(* CODESYS project XLH_base_START_01_00.project
   Description: Receives some incoming messages and echoes them with CAN-ID +1
   Title: CAN Bus API Example
   Version: 1.0.0.0
   Company: 3S - Smart Software Solutions GmbH
   Author: 3S - Smart Software Solutions GmbH

Project tree, tasks and I/O mapping:
  XLH_base : CODESYS Control for Raspberry Pi SL, CODESYS, order no. 2302000009, version 4.12.0.0
    application app
      libraries: Standard, 3.5.18.0 (System); Memory, * (3S - Smart Software Solutions GmbH); Util, 3.5.19.0 (System); VisuDialogs, * (System); CAA Tick Extern, 3.5.17.0 (CAA Technical Workgroup); SysTime, 3.5.17.0 (System); CmpIecTask, * (System); xemax Bibliothek, 0.10 (xemax ag)
      task MAIN_TASK (cyclic, interval 20 ms, priority 0) calls MAIN, io
      task VISU_TASK (cyclic, interval 100 ms, priority 31) calls VisuElems.Visu_Prg
      program io [ST]
      visualisation VISU
      program MAIN [ST]
    SoftMotion General Axis Pool
    GPIOs_A_B : GPIOs B+/Pi2, CODESYS, version 4.12.0.0
        input  app.io.bSw1 : BOOL  // digital inputs (GPIO0..GPIO31).Bit4
        input  app.io.bSw2 : BOOL  // digital inputs (GPIO0..GPIO31).Bit5
        input  app.io.bSw3 : BOOL  // digital inputs (GPIO0..GPIO31).Bit6
        input  app.io.bSw4 : BOOL  // digital inputs (GPIO0..GPIO31).Bit12
        input  app.io.bSw5 : BOOL  // digital inputs (GPIO0..GPIO31).Bit13
        input  app.io.bSw6 : BOOL  // digital inputs (GPIO0..GPIO31).Bit16
        input  app.io.bSw7 : BOOL  // digital inputs (GPIO0..GPIO31).Bit17
        input  app.io.bSw8 : BOOL  // digital inputs (GPIO0..GPIO31).Bit19
        output app.io.bLed1 : BOOL  // digital outputs (GPIO0..GPIO31).Bit20
        output app.io.bLed2 : BOOL  // digital outputs (GPIO0..GPIO31).Bit21
        output app.io.bLed3 : BOOL  // digital outputs (GPIO0..GPIO31).Bit22
        output app.io.bLed4 : BOOL  // digital outputs (GPIO0..GPIO31).Bit23
        output app.io.bLed5 : BOOL  // digital outputs (GPIO0..GPIO31).Bit24
        output app.io.bLed6 : BOOL  // digital outputs (GPIO0..GPIO31).Bit26
        output app.io.bLed7 : BOOL  // digital outputs (GPIO0..GPIO31).Bit27
        unmapped channels: digital inputs (GPIO0..GPIO31), digital outputs (GPIO0..GPIO31)
    Onewire
    Camera device
      <Leer>
    SPI
    I²C
    Ethernet : Ethernet, CODESYS, version 4.2.0.0
        settings: IPAddress = [127,0,0,1]; SubnetMask = [255,0,0,0]; GatewayAddress = [0,0,0,0]; NetworkInterfaceName = 'lo'; NetworkInterfaceName = "lo"; SaveCommunicationSettings = FALSE
      ModbusTCP_Slave_OLED_Port_503 : ModbusTCP Slave Device, CODESYS, version 4.3.0.0
          settings: Port = 503
          output app.io.oled.awToOled : ARRAY[0..32] OF WORD  // Ausgänge
          unmapped channels: Eingänge
  libraries: VisuSymbols, 4.5.0.0 (System); DepictorBase, 1.0.5.0 (3S - Smart Software Solutions GmbH)
  text list GlobalTextList
*)

// XLH_base/app/MAIN
PROGRAM MAIN
VAR
	vVersionPlc: VERSION;
	sVersionPlc: STRING(255);
	vVersionLib: VERSION;
	sVersionLib: STRING(255);
END_VAR

// Version Bibliothex xemax
vVersionPlc.uiMajor := 1;
vVersionPlc.uiMinor := 0;
sVersionPlc := CONCAT(TO_STRING(TO_UINT(vVersionPlc.uiMajor)), CONCAT('.', (TO_STRING(TO_UINT(vVersionPlc.uiMinor)))));
vVersionLib := xemax.GetLibVersion();
sVersionLib := CONCAT(TO_STRING(TO_UINT(vVersionLib.uiMajor)), CONCAT('.', (TO_STRING(TO_UINT(vVersionLib.uiMinor)))));

(*
==================================================================================================
Login Codesys in die XLH - SPS 
user: pi
pw: pi
==================================================================================================
Webvisualisierung
http://ip:8080/webvisu.htm
- bei einer Verbindung via USB: http://192.168.31.31:8080/webvisu.htm
- bei einer Verbindung via USB-RJ45-Adapter: http://192.168.1.31:8080/webvisu.htm
==================================================================================================
OPC-UA
anonymous (ohne Benutzer und Passwort)
opc.tcp://192.168.31.31:4840
==================================================================================================
RGB-Matrix
im aktuellen BETA-Status kann die Matrix via REST-API angesteurt werden
https://de.wikipedia.org/wiki/Representational_State_Transfer
http://192.168.1.31:8077/rgb/0/1/0

Weiter geplant ist eine Umsetzung zur Ansteuerung der RGB Matrix als IoT Device via MQTT
 
Die Integration in Codesys ist noch ausstehend 
==================================================================================================
Login XLH - Linuxumgebung via Putty
user: pi
pw: pi
==================================================================================================
Konfiguration WiFi 
sudo nano /etc/wpa_supplicant/wpa_supplicant.conf

network={
        ssid="abc"
        psk="def"
        key_mgmt=WPA-PSK
}
==================================================================================================
statische IP USB-Ethernet-Erweiterung: 
sudo nano /etc/dhcpcd.conf
# profile static_eth0
...
==================================================================================================
*)

END_PROGRAM

// XLH_base/app/io
PROGRAM io
VAR_INPUT			
	bLed1: BOOL;
	bLed2: BOOL;
	bLed3: BOOL;
	bLed4: BOOL;
	bLed5: BOOL;
	bLed6: BOOL;
	bLed7: BOOL;	
	oled: OLED;
END_VAR
VAR_OUTPUT
	bSw1: BOOL;
	bSw2: BOOL;
	bSw3: BOOL;
	bSw4: BOOL;
	bSw5: BOOL;
	bSw6: BOOL;
	bSw7: BOOL;
	bSw8: BOOL;
END_VAR
VAR
END_VAR

xemax.LOCAL_TIME_AND_TIME_ZONE();
xemax.TASK_INFO();
oled();

END_PROGRAM

// XLH_base/app/VISU
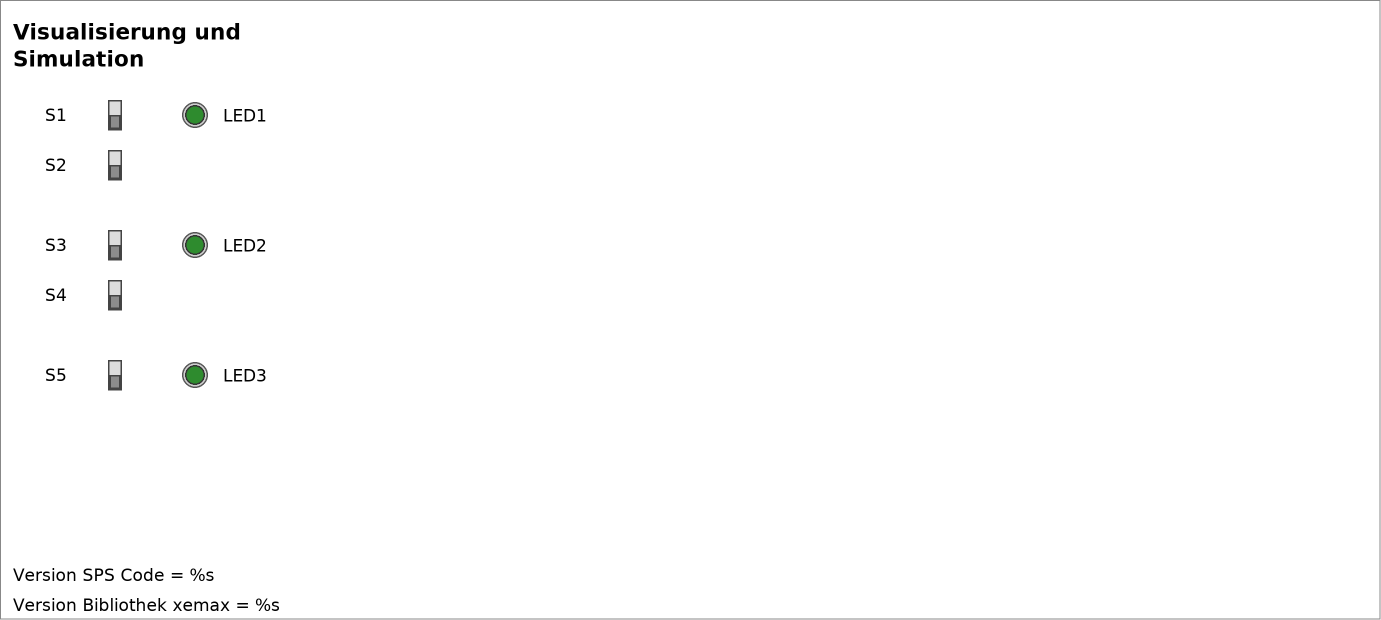
VISUALIZATION VISU  // 1381x620
    Rectangle (220,90 81x51), "LED1"
    Rectangle (10,10 461x71), "Visualisierung und Simulation"
    Line (1380,270)
    DipSwitch (80,100 70x30), variable: io.bSw1, behaviour: TOGGLE, style: Switch-DipSwitch-Gray
    Rectangle (20,90 50x50), "S1"
    Lamp1 (180,100 30x30), variable: io.bLed1, style: Lamp-Lamp1-Green
    Rectangle (10,560 291x30), "Version SPS Code = %s", text variable: MAIN.sVersionPlc
    Rectangle (10,590 291x30), "Version Bibliothek xemax = %s", text variable: MAIN.sVersionLib
    Rectangle (20,140 50x50), "S2"
    DipSwitch (80,150 70x30), variable: io.bSw2, behaviour: TOGGLE, style: Switch-DipSwitch-Gray
    Rectangle (220,220 81x51), "LED2"
    DipSwitch (80,230 70x30), variable: io.bSw3, behaviour: TOGGLE, style: Switch-DipSwitch-Gray
    Rectangle (20,220 50x50), "S3"
    Lamp1 (180,230 30x30), variable: io.bLed2, style: Lamp-Lamp1-Green
    Rectangle (20,270 50x50), "S4"
    DipSwitch (80,280 70x30), variable: io.bSw4, behaviour: TOGGLE, style: Switch-DipSwitch-Gray
    Rectangle (220,350 81x51), "LED3"
    DipSwitch (80,360 70x30), variable: io.bSw5, behaviour: TOGGLE, style: Switch-DipSwitch-Gray
    Rectangle (20,350 50x50), "S5"
    Lamp1 (180,360 30x30), variable: io.bLed3, style: Lamp-Lamp1-Green
END_VISUALIZATION
